ABB RAPID module: aRob3HC16.mod

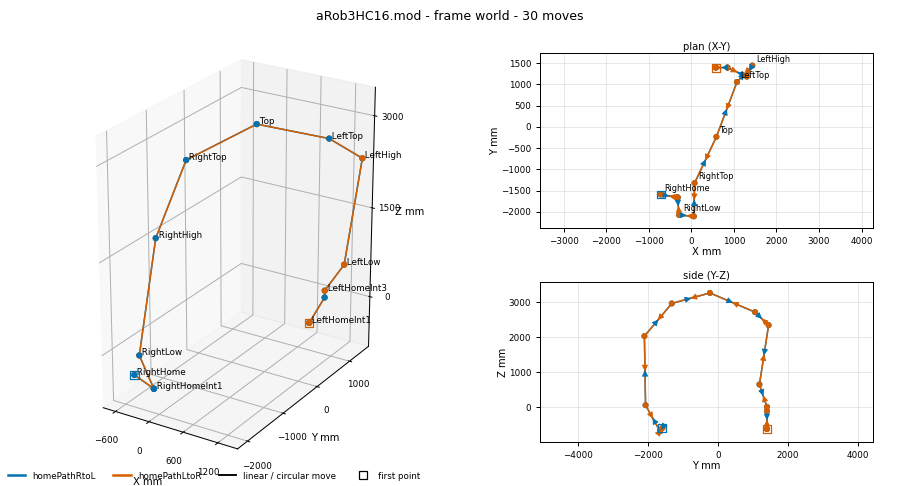
[picture p0: tool path of aRob3HC16.mod in frame world, 30 of 30 moves have a stored position in this frame; points joined in program order, loops and branches not executed]
MODULE TestHomeCircuit3

    CONST robtarget LeftHome:=[[576.85,1394.56,-612.51],[0.509771,0.539227,-0.479592,-0.468359],[0,-2,0,1],[9E+09,9E+09,9E+09,9E+09,9E+09,9E+09]];
	CONST robtarget LeftHomeInt1:=[[576.85,1394.56,-612.51],[0.114649,0.144984,-0.689844,-0.699965],[0,-1,0,1],[9E+09,9E+09,9E+09,9E+09,9E+09,9E+09]];
	CONST robtarget LeftHomeInt2:=[[848.55,1394.57,-101.1],[0.156024,0.241541,0.825171,0.486219],[0,0,0,1],[9E+09,9E+09,9E+09,9E+09,9E+09,9E+09]];
	CONST robtarget LeftHomeInt3:=[[848.55,1394.57,18.07],[0.262988,0.312453,0.79354,0.451115],[0,0,0,1],[9E+09,9E+09,9E+09,9E+09,9E+09,9E+09]];
	CONST robtarget LeftHomeInt4:=[[1167.86,1394.59,188.72],[0.267191,0.437633,0.678207,0.526424],[0,0,1,1],[9E+09,9E+09,9E+09,9E+09,9E+09,9E+09]];

	CONST robtarget LeftLow:=[[1304.39,1181.14,656.35],[0.041734,0.725074,0.686734,0.030393],[0,1,-1,1],[9E+09,9E+09,9E+09,9E+09,9E+09,9E+09]];

	CONST robtarget LeftHigh:=[[1434.23,1442.35,2349.62],[0.033258,0.713022,0.699985,0.022699],[0,1,-1,1],[9E+09,9E+09,9E+09,9E+09,9E+09,9E+09]];

	CONST robtarget LeftTop:=[[1073,1056.21,2720.53],[0.360733,0.617475,0.611089,0.339363],[0,1,-1,1],[9E+09,9E+09,9E+09,9E+09,9E+09,9E+09]] ;
    CONST robtarget Top:=[[589.15,-232.43,3269.58],[0.573092,0.594807,0.417225,0.37907],[-1,2,-2,1],[9E+09,9E+09,9E+09,9E+09,9E+09,9E+09]];


	CONST robtarget RightTop:=[[76.05,-1322.06,2968.83],[0.37033,0.788742,0.472236,0.133176],[-2,2,-2,1],[9E+09,9E+09,9E+09,9E+09,9E+09,9E+09]];
    CONST robtarget RightHigh:=[[61.04,-2103.13,2035.96],[0.116709,0.878807,0.459988,0.04988],[-1,2,-2,1],[9E+09,9E+09,9E+09,9E+09,9E+09,9E+09]];
    CONST robtarget RightLow:=[[-287.84,-2070.36,65.02],[0.026826,0.901845,0.431199,0.004971],[-2,2,-2,1],[9E+09,9E+09,9E+09,9E+09,9E+09,9E+09]];

	CONST robtarget RightHomeInt4:=[[-322.21,-1658.14,-677.51],[0.334256,0.336793,0.589508,0.6537],[-2,2,-3,1],[9E+09,9E+09,9E+09,9E+09,9E+09,9E+09]];
   	CONST robtarget RightHomeInt3:=[[-322.21,-1658.14,-677.51],[0.334256,0.336793,0.589508,0.6537],[-2,2,-3,1],[9E+09,9E+09,9E+09,9E+09,9E+09,9E+09]];
	CONST robtarget RightHomeInt2:=[[-322.21,-1658.14,-677.51],[0.334256,0.336793,0.589508,0.6537],[-2,2,-3,1],[9E+09,9E+09,9E+09,9E+09,9E+09,9E+09]];
	CONST robtarget RightHomeInt1:=[[-322.21,-1658.14,-677.51],[0.334256,0.336793,0.589508,0.6537],[-2,2,-3,1],[9E+09,9E+09,9E+09,9E+09,9E+09,9E+09]];
    CONST robtarget RightHome:=[[-721.44,-1589.68,-584.17],[0.312267,0.264728,0.705871,0.578062],[-2,2,-4,1],[9E+09,9E+09,9E+09,9E+09,9E+09,9E+09]];

    PROC Main()

        homePathLtoR;
		homePathRtoL;

    ENDPROC


    PROC homePathRtoL()

        MoveL RightHome,v100,z100,tool0\WObj:=wobj0;
		MoveL RightHomeInt1,v100,z100,tool0\WObj:=wobj0;
		MoveL RightHomeInt2,v100,z100,tool0\WObj:=wobj0;
		MoveL RightHomeInt3,v100,z100,tool0\WObj:=wobj0;
        MoveL RightLow,v100,z100,tool0\WObj:=wobj0;
        MoveL RightHigh,v100,z100,tool0\WObj:=wobj0;
        MoveL RightTop,v100,z100,tool0\WObj:=wobj0;

		MoveL Top,v100,z100,tool0\WObj:=wobj0;

		MoveL LeftTop,v100,z100,tool0\WObj:=wobj0;
        MoveL LeftHigh,v100,z100,tool0\WObj:=wobj0;
        MoveL LeftLow,v100,z100,tool0\WObj:=wobj0;

		MoveL LeftHomeInt3,v100,z100,tool0\WObj:=wobj0;
		MoveL LeftHomeInt2,v100,z100,tool0\WObj:=wobj0;
		MoveL LeftHomeInt1,v100,z100,tool0\WObj:=wobj0;
        MoveL LeftHome,v100,z100,tool0\WObj:=wobj0;

    ENDPROC

	PROC homePathLtoR()

		MoveL LeftHome,v100,z100,tool0\WObj:=wobj0;
		MoveL LeftHomeInt1,v100,z100,tool0\WObj:=wobj0;
		MoveL LeftHomeInt2,v100,z100,tool0\WObj:=wobj0;
		MoveL LeftHomeInt3,v100,z100,tool0\WObj:=wobj0;


		MoveL LeftLow,v100,z100,tool0\WObj:=wobj0;
        MoveL LeftHigh,v100,z100,tool0\WObj:=wobj0;
		MoveL LeftTop,v100,z100,tool0\WObj:=wobj0;

		MoveL Top,v100,z100,tool0\WObj:=wobj0;

		MoveL RightTop,v100,z100,tool0\WObj:=wobj0;
		MoveL RightHigh,v100,z100,tool0\WObj:=wobj0;
		MoveL RightLow,v100,z100,tool0\WObj:=wobj0;

		MoveL RightHomeInt3,v100,z100,tool0\WObj:=wobj0;
		MoveL RightHomeInt2,v100,z100,tool0\WObj:=wobj0;
		MoveL RightHomeInt1,v100,z100,tool0\WObj:=wobj0;
		MoveL RightHome,v100,z100,tool0\WObj:=wobj0;

	ENDPROC







ENDMODULE
